TYPE ST_AxisStruct :
STRUCT
    stControl: ST_AxisControl;
    stStatus: ST_AxisStatus;
    stConfig: ST_AxisConfig;
    stError: ST_AxisError;
    stInputs: ST_AxisInputs;
    stDescription: ST_AxisDescription;
	stHomingConfig : ST_AxisHomingConfig;
	stSpg : ST_AxisSPG;
    //The NC axis link to the hardware that is controlling
    Axis: AXIS_REF;
	Commissioning : BOOL :=FALSE;
END_STRUCT
END_TYPE

(* stored: Version 1.1.0.1, ProductVersion 3.1.4026.18
   DUT ST_AxisStruct: Id {9732127f-85ab-48d1-a591-d13402fe3665} *)
